TYPE ST_CURING_STATION_SETTINGS :
STRUCT
END_STRUCT
END_TYPE

(* stored: Version 1.1.0.1
   DUT ST_CURING_STATION_SETTINGS: Id {8b058acc-cb09-444a-8198-745c1eee0bb6} *)
